Staubli VAL3: DataBase.pjx

--- DataBase.pjx ---
Parameters version=s7.7 stackSize=5000 millimeterUnit=true
Program file=start.pgx
Program file=stop.pgx
Data file=DataBase.dtx

--- DataBase.dtx ---
public bool bAirOn
public bool bAlarm
public bool bDebugMode
public bool bExtraContrAxis
public bool bFollowOn
public bool bGasChoose
public bool bIOControl = true
public bool bIOStart
public bool bIsHome
public bool bKeyIO[3]
public bool bLaserOn
public bool bMoveTask
public bool bMultiNormal
public bool bMutexAxis
public bool bPowerOn
public bool bSaveTrajPoint
public bool bSingleAxisMode = true
public bool bStopPoll
public bool bStopSimul = true
public bool bThickPlatPunch
public bool bThickPlate
public bool bUpload
public bool bWaitFollowDone
public bool bWorldMove = true
public bool bWpFinishIOOut
public frame fFrame = {fatherId=world[0]}
public frame fJogContext = {fatherId=world[0]}
public frame fOffset = {fatherId=world[0]}
public jointRx jCurrentJoint = {j1=-0.537933, j2=20.526668, j3=117.407786, j4=-3.817874, j5=-48.245361, j6=2.958515}
public mdesc mJHome = {tmax=166.666667, blend=off}
mdesc mNomSpeed
public num n1AxisOffset = 0.1
public num nActionID = 0.258567
public num nArrayCutAction[2]
public num nArrayX = 1
public num nArrayY = 1
public num nArrayZ = 1
public num nAsysAxisPer = 0.008
public num nAvgCutSpeed = 177.53368
public num nAxisOffset[2]
public num nCutLength = 393.307878
public num nCutTime = 3.117
public num nCycleCount
public num nCycleIndex
public num nCycleMode
public num nCycleTime = 36.639
public num nDebugData
public num nID
public num nInterfaceType = 7
public num nPartMove[3]
public num nPointType
public num nPollTime = 0.028
public num nPresetData[5]
  [1] = -100
public num nProductCount
public num nProductIndex
public num nRemoteProduct
public num nRobotSpeed
public num nSpeedPercent = 1
public num nTestData
public num nToolMode = 1
public num nTrajIndex = 1
public num nVersion = 3
public num nWeldActionId
public num nWeldEndOffset = 10
public num nWeldEndStart
public num nWeldEndTime = 9217.537
public num nWeldStartTime
public num nWorkPlaceButto = -1
public num nWorkPlaceCount
public num nWorkPlaceIndex
public num nWpMutiCount[10]
public num nWpProduct[5]
public pointRx pCurrentPoint = {x=1238.856806, y=-1.545091, z=-197.49862, rx=0.00299859, ry=179.999837, rz=-0.00317733, shoulder=lefty, elbow=epositive, wrist=wnegative, fatherId=world[0]}
string sCustom
public string sProductName[10]
  [0] = "3d"
  [1] = "test20150408"
public string sSoftWareTime = "2015_02_03"
public string sVersion[8]
  [0] = "s7.9 - Dec 10 2015 - 10:53:01"
  [1] = "rx160l-S1"
  [2] = "floor"
  [3] = "?"
public trsf trOffset[3]
public trsf trTeachTemp = {z=300, rx=15}
